FUNCTION alg_a_TledQ1: BOOL
VAR_INPUT
    state: STATE;
END_VAR

alg_a_TledQ1 := (state.dvar_M_led1) = (elit_On);

END_FUNCTION

(* stored: ProductVersion 3.1.0.18, Version 1.1.0.1 *)
